(*This structure is for a single Alarm*)
TYPE Alarm_Type :
STRUCT

	State: BOOL:=0; (*Bit that tracks error state; 0=okay, 1=active*)
	Override: BOOL:=0; (*Error Override Bit*)
	Name: STRING:=''; (*Array for error names*)

END_STRUCT
END_TYPE

(* stored: Version 1.1.0.1, ProductVersion 3.1.0.38
   DUT ALARM_TYPE: Id {c3ffcf74-49b4-46c6-bdcc-31731eeb722c} *)
